(* Logix 5000 project; controller FRCFMS vendor 1 type 14 code 150 rev 33.11; software revision 33.00; part 3 of 3 *)
(* tags used below, declared in another part *)
   CMD_END : DINT;
   CMD_IN : DINT;
   CMD_LEN : DINT;
   CMD_LEN1 : INT;
   CMD_LEN2 : INT;
   CMD_START : DINT;
   Conn_Open : BOOL[32];
   EX_CMD : INT;
   EX_CODE : INT;
   MB_Resp_Data : STR_462;
   Modbus_Byte_cnt : INT;
   Modbus_Cmd_String : STR_462;
   Modbus_Ret_CMD : STRING;
   Modbus_Ret_len : STRING;
   Next_Write : BOOL[32];
   ONS : BOOL[64];
   ONS_B : BOOL[32];
   ONS_ERR : BOOL[32];
   RG_4x_Pos : DINT;
   RW_Instance : INT[20];
   RW_Select : DINT;
   String_Pos : INT;
   Valid : BOOL[32];
   Valid_CMD : BOOL[32];
   Valid_End : BOOL;
   Valid_Len : BOOL;
   Valid_Len_16 : BOOL;
   Valid_Start_Addr : BOOL;
   MBTI_Read_Data_MSG_00 : MESSAGE;
   MBTI_Read_Data_MSG_01 : MESSAGE;
   MBTI_Read_Data_MSG_02 : MESSAGE;
   MBTI_Read_Data_MSG_03 : MESSAGE;
   MBTI_Read_Data_MSG_04 : MESSAGE;
   MBTI_Read_Data_MSG_05 : MESSAGE;
   MBTI_Read_Data_MSG_06 : MESSAGE;
   MBTI_Read_Data_MSG_07 : MESSAGE;
   MBTI_Read_Data_MSG_08 : MESSAGE;
   MBTI_Read_Data_MSG_09 : MESSAGE;
   MBTI_Read_Done : BOOL[32];
   MBTI_Read_Resp : READ_RESP_STR[10];
   MBTI_Write_Data_MSG_00 : MESSAGE;
   MBTI_Write_Data_MSG_01 : MESSAGE;
   MBTI_Write_Data_MSG_02 : MESSAGE;
   MBTI_Write_Data_MSG_03 : MESSAGE;
   MBTI_Write_Data_MSG_04 : MESSAGE;
   MBTI_Write_Data_MSG_05 : MESSAGE;
   MBTI_Write_Data_MSG_06 : MESSAGE;
   MBTI_Write_Data_MSG_07 : MESSAGE;
   MBTI_Write_Data_MSG_08 : MESSAGE;
   MBTI_Write_Data_MSG_09 : MESSAGE;
   MBTI_Write_Data_Out : WRT_DATA[10];
   MBTU_MB_4xx : INT[100];
(* ModbusSlaveTCP, continued *)

ROUTINE SUB_Resp_Str_WORD   (* ladder *)
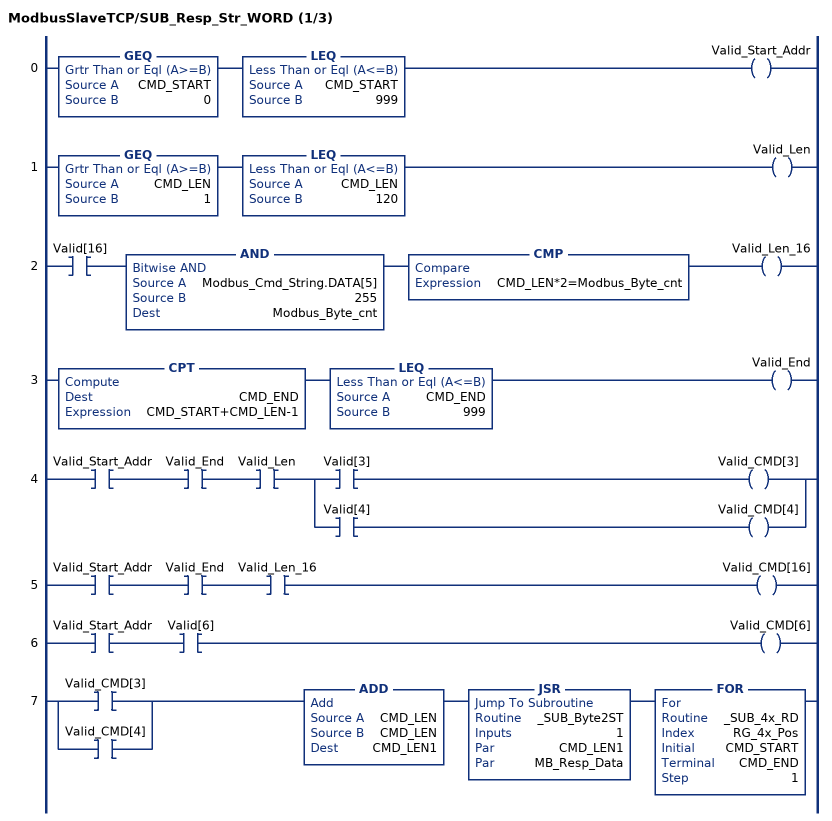
   0: GEQ(CMD_START,0)LEQ(CMD_START,999)OTE(Valid_Start_Addr);
   1: GEQ(CMD_LEN,1)LEQ(CMD_LEN,120)OTE(Valid_Len);
   2: XIC(Valid[16])AND(Modbus_Cmd_String.DATA[5],255,Modbus_Byte_cnt)CMP(CMD_LEN*2=Modbus_Byte_cnt)OTE(Valid_Len_16);
   3: CPT(CMD_END,CMD_START+CMD_LEN-1)LEQ(CMD_END,999)OTE(Valid_End);
   4: XIC(Valid_Start_Addr)XIC(Valid_End)XIC(Valid_Len)[XIC(Valid[3]) OTE(Valid_CMD[3]) ,XIC(Valid[4]) OTE(Valid_CMD[4]) ];
   5: XIC(Valid_Start_Addr)XIC(Valid_End)XIC(Valid_Len_16)OTE(Valid_CMD[16]);
   6: XIC(Valid_Start_Addr)XIC(Valid[6])OTE(Valid_CMD[6]);
   7: [XIC(Valid_CMD[3]) ,XIC(Valid_CMD[4]) ]ADD(CMD_LEN,CMD_LEN,CMD_LEN1)JSR(_SUB_Byte2ST,1,CMD_LEN1,MB_Resp_Data)FOR(_SUB_4x_RD,RG_4x_Pos,CMD_START,CMD_END,1);
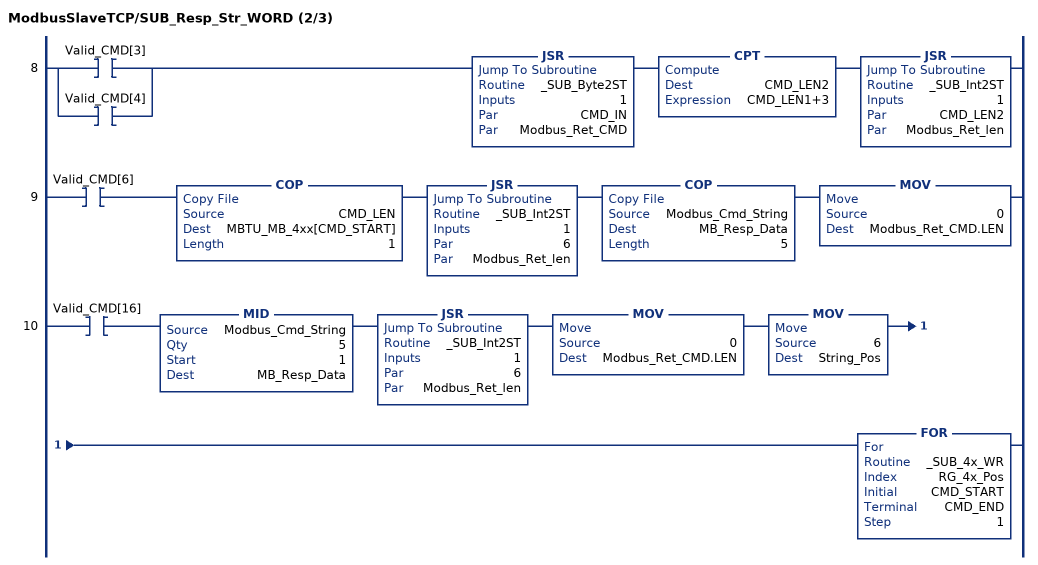
   8: [XIC(Valid_CMD[3]) ,XIC(Valid_CMD[4]) ]JSR(_SUB_Byte2ST,1,CMD_IN,Modbus_Ret_CMD)CPT(CMD_LEN2,CMD_LEN1+3)JSR(_SUB_Int2ST,1,CMD_LEN2,Modbus_Ret_len);
   9: XIC(Valid_CMD[6])COP(CMD_LEN,MBTU_MB_4xx[CMD_START],1)JSR(_SUB_Int2ST,1,6,Modbus_Ret_len)COP(Modbus_Cmd_String,MB_Resp_Data,5)MOV(0,Modbus_Ret_CMD.LEN);
   10: XIC(Valid_CMD[16])MID(Modbus_Cmd_String,5,1,MB_Resp_Data)JSR(_SUB_Int2ST,1,6,Modbus_Ret_len)MOV(0,Modbus_Ret_CMD.LEN)MOV(6,String_Pos)FOR(_SUB_4x_WR,RG_4x_Pos,CMD_START,CMD_END,1);
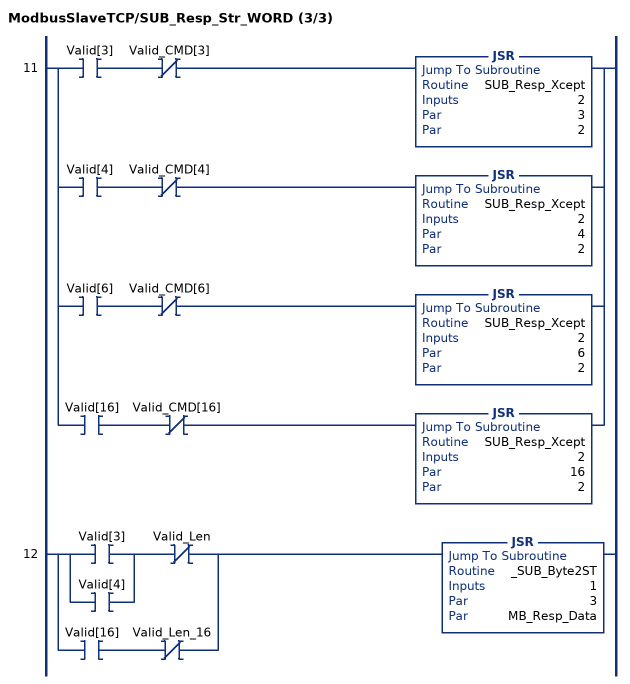
   11: [XIC(Valid[3]) XIO(Valid_CMD[3]) JSR(SUB_Resp_Xcept,2,3,2) ,XIC(Valid[4]) XIO(Valid_CMD[4]) JSR(SUB_Resp_Xcept,2,4,2) ,XIC(Valid[6]) XIO(Valid_CMD[6]) JSR(SUB_Resp_Xcept,2,6,2) ,XIC(Valid[16]) XIO(Valid_CMD[16]) JSR(SUB_Resp_Xcept,2,16,2) ];
   12: [[XIC(Valid[3]) ,XIC(Valid[4]) ] XIO(Valid_Len) ,XIC(Valid[16]) XIO(Valid_Len_16) ]JSR(_SUB_Byte2ST,1,3,MB_Resp_Data);
END_ROUTINE

ROUTINE SUB_Resp_Xcept   (* ladder *)
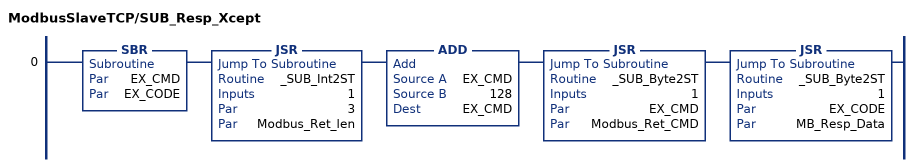
   0: SBR(EX_CMD,EX_CODE)JSR(_SUB_Int2ST,1,3,Modbus_Ret_len)ADD(EX_CMD,128,EX_CMD)JSR(_SUB_Byte2ST,1,EX_CMD,Modbus_Ret_CMD)JSR(_SUB_Byte2ST,1,EX_CODE,MB_Resp_Data);
END_ROUTINE

ROUTINE SUB_RW_Messages   (* ladder *)
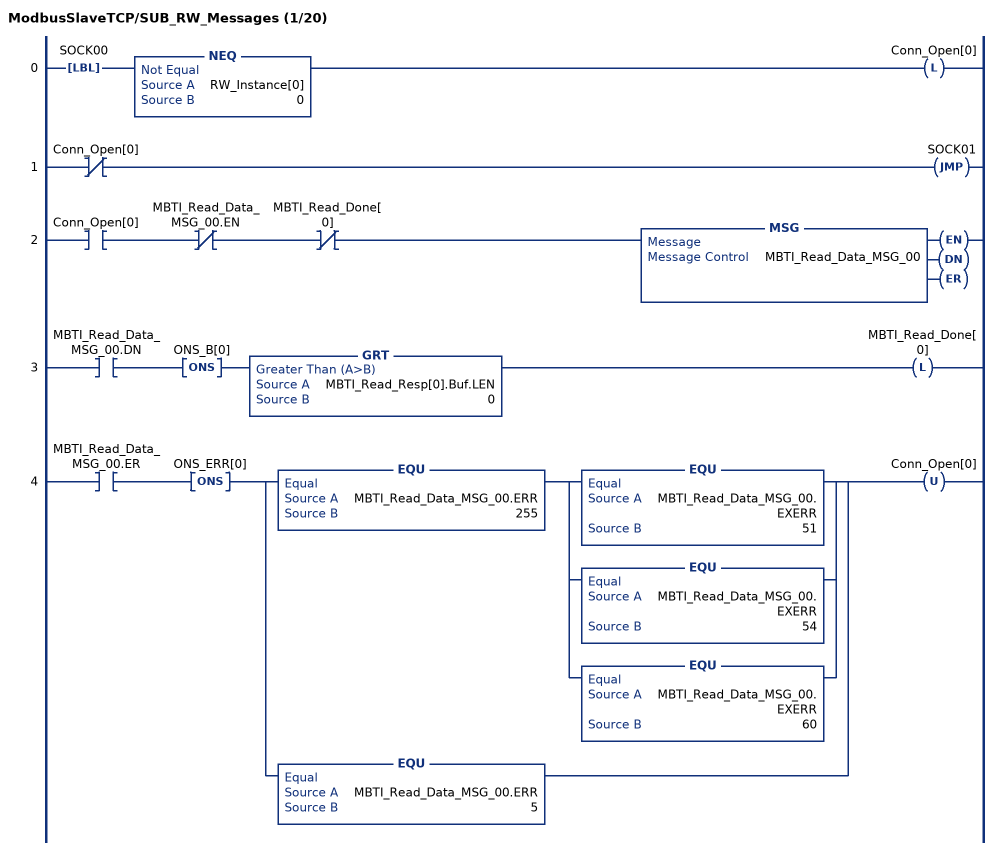
   0: LBL(SOCK00)NEQ(RW_Instance[0],0)OTL(Conn_Open[0]);
   1: XIO(Conn_Open[0])JMP(SOCK01);
   2: XIC(Conn_Open[0])XIO(MBTI_Read_Data_MSG_00.EN)XIO(MBTI_Read_Done[0])MSG(MBTI_Read_Data_MSG_00);
   3: XIC(MBTI_Read_Data_MSG_00.DN)ONS(ONS_B[0])GRT(MBTI_Read_Resp[0].Buf.LEN,0)OTL(MBTI_Read_Done[0]);
   4: XIC(MBTI_Read_Data_MSG_00.ER)ONS(ONS_ERR[0])[EQU(MBTI_Read_Data_MSG_00.ERR,255) [EQU(MBTI_Read_Data_MSG_00.EXERR,51) ,EQU(MBTI_Read_Data_MSG_00.EXERR,54) ,EQU(MBTI_Read_Data_MSG_00.EXERR,60) ] ,EQU(MBTI_Read_Data_MSG_00.ERR,5) ]OTU(Conn_Open[0]);
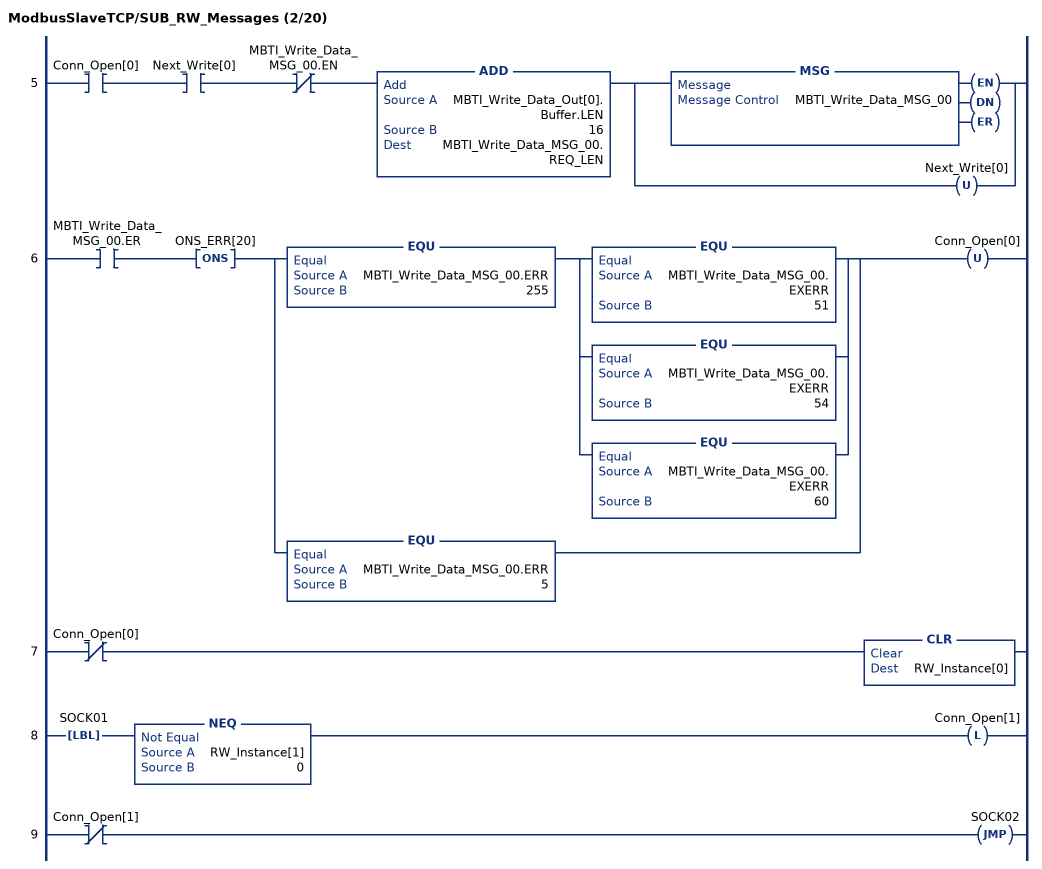
   5: XIC(Conn_Open[0])XIC(Next_Write[0])XIO(MBTI_Write_Data_MSG_00.EN)ADD(MBTI_Write_Data_Out[0].Buffer.LEN,16,MBTI_Write_Data_MSG_00.REQ_LEN)[MSG(MBTI_Write_Data_MSG_00) ,OTU(Next_Write[0]) ];
   6: XIC(MBTI_Write_Data_MSG_00.ER)ONS(ONS_ERR[20])[EQU(MBTI_Write_Data_MSG_00.ERR,255) [EQU(MBTI_Write_Data_MSG_00.EXERR,51) ,EQU(MBTI_Write_Data_MSG_00.EXERR,54) ,EQU(MBTI_Write_Data_MSG_00.EXERR,60) ] ,EQU(MBTI_Write_Data_MSG_00.ERR,5) ]OTU(Conn_Open[0]);
   7: XIO(Conn_Open[0])CLR(RW_Instance[0]);
   8: LBL(SOCK01)NEQ(RW_Instance[1],0)OTL(Conn_Open[1]);
   9: XIO(Conn_Open[1])JMP(SOCK02);
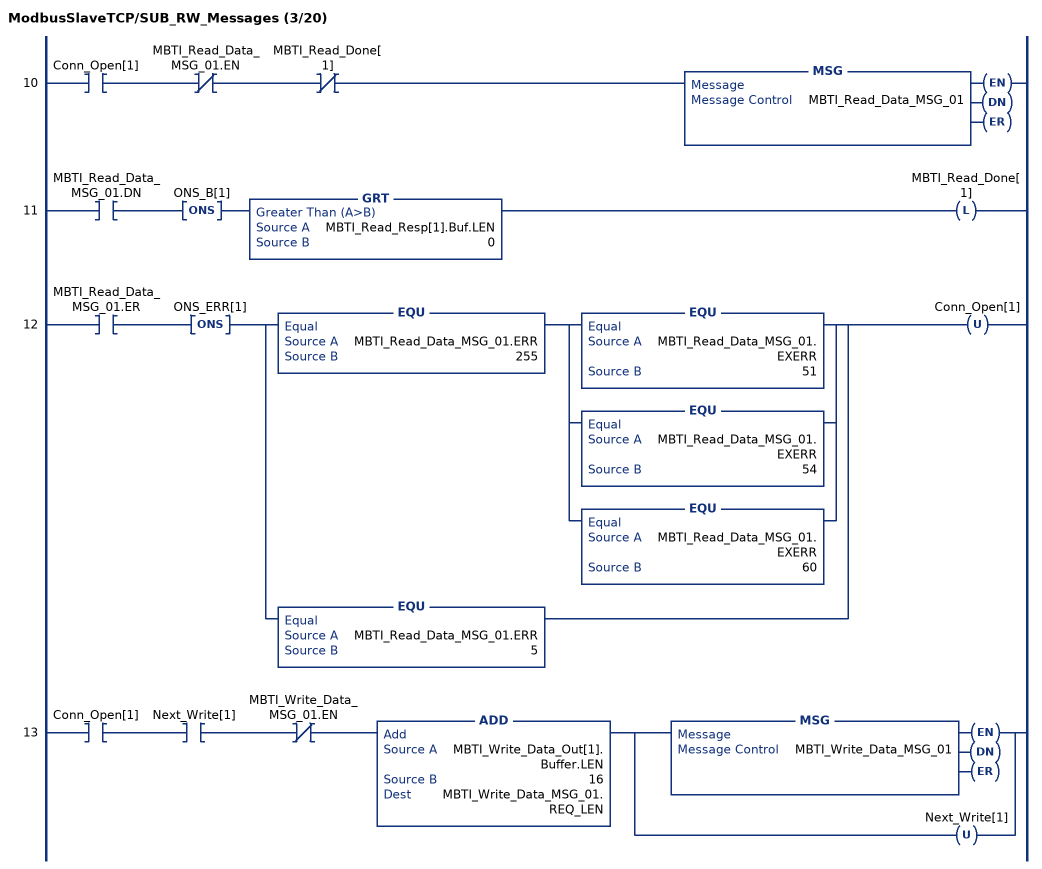
   10: XIC(Conn_Open[1])XIO(MBTI_Read_Data_MSG_01.EN)XIO(MBTI_Read_Done[1])MSG(MBTI_Read_Data_MSG_01);
   11: XIC(MBTI_Read_Data_MSG_01.DN)ONS(ONS_B[1])GRT(MBTI_Read_Resp[1].Buf.LEN,0)OTL(MBTI_Read_Done[1]);
   12: XIC(MBTI_Read_Data_MSG_01.ER)ONS(ONS_ERR[1])[EQU(MBTI_Read_Data_MSG_01.ERR,255) [EQU(MBTI_Read_Data_MSG_01.EXERR,51) ,EQU(MBTI_Read_Data_MSG_01.EXERR,54) ,EQU(MBTI_Read_Data_MSG_01.EXERR,60) ] ,EQU(MBTI_Read_Data_MSG_01.ERR,5) ]OTU(Conn_Open[1]);
   13: XIC(Conn_Open[1])XIC(Next_Write[1])XIO(MBTI_Write_Data_MSG_01.EN)ADD(MBTI_Write_Data_Out[1].Buffer.LEN,16,MBTI_Write_Data_MSG_01.REQ_LEN)[MSG(MBTI_Write_Data_MSG_01) ,OTU(Next_Write[1]) ];
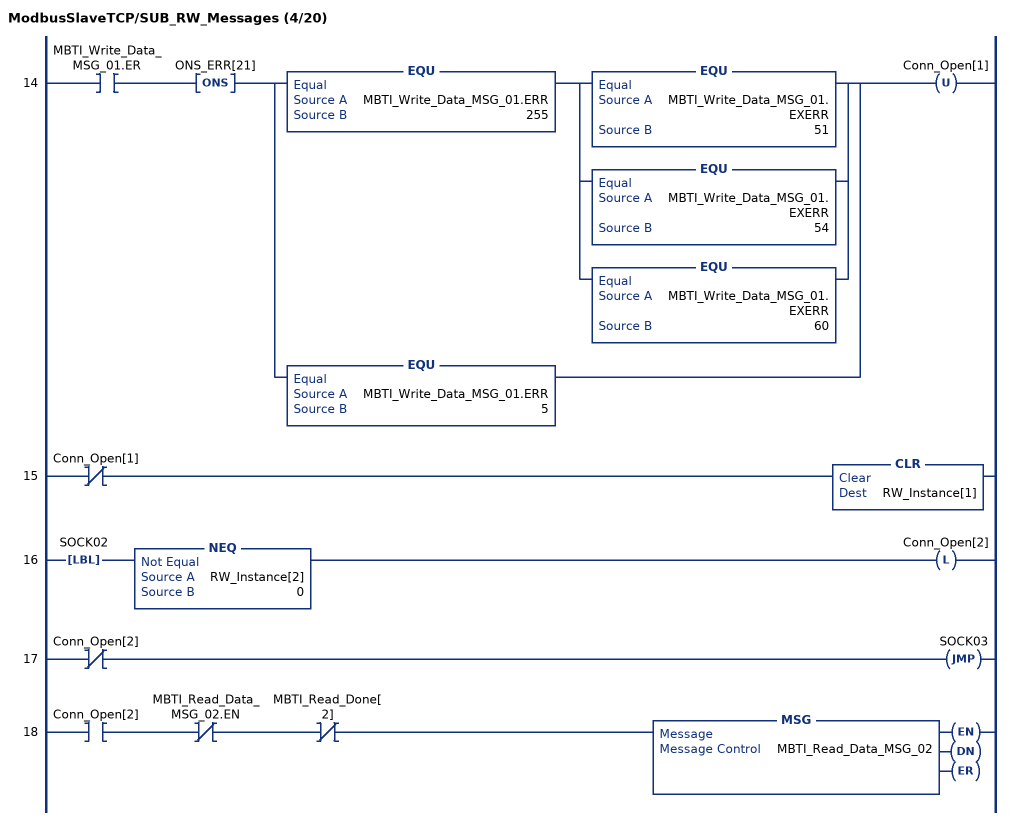
   14: XIC(MBTI_Write_Data_MSG_01.ER)ONS(ONS_ERR[21])[EQU(MBTI_Write_Data_MSG_01.ERR,255) [EQU(MBTI_Write_Data_MSG_01.EXERR,51) ,EQU(MBTI_Write_Data_MSG_01.EXERR,54) ,EQU(MBTI_Write_Data_MSG_01.EXERR,60) ] ,EQU(MBTI_Write_Data_MSG_01.ERR,5) ]OTU(Conn_Open[1]);
   15: XIO(Conn_Open[1])CLR(RW_Instance[1]);
   16: LBL(SOCK02)NEQ(RW_Instance[2],0)OTL(Conn_Open[2]);
   17: XIO(Conn_Open[2])JMP(SOCK03);
   18: XIC(Conn_Open[2])XIO(MBTI_Read_Data_MSG_02.EN)XIO(MBTI_Read_Done[2])MSG(MBTI_Read_Data_MSG_02);
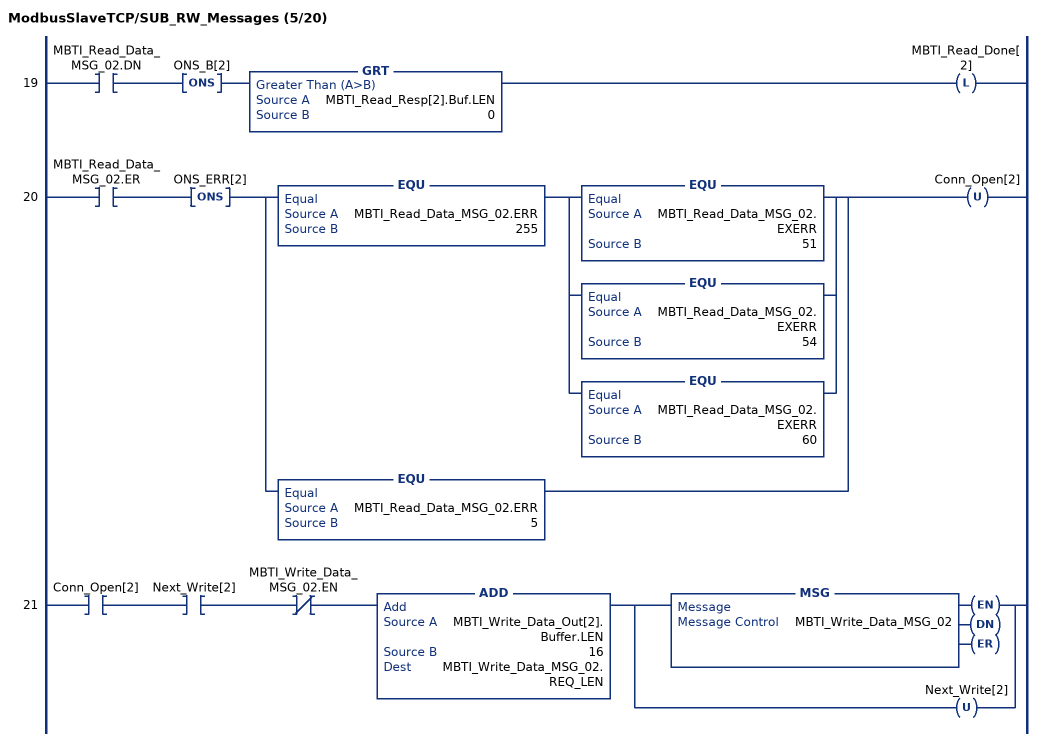
   19: XIC(MBTI_Read_Data_MSG_02.DN)ONS(ONS_B[2])GRT(MBTI_Read_Resp[2].Buf.LEN,0)OTL(MBTI_Read_Done[2]);
   20: XIC(MBTI_Read_Data_MSG_02.ER)ONS(ONS_ERR[2])[EQU(MBTI_Read_Data_MSG_02.ERR,255) [EQU(MBTI_Read_Data_MSG_02.EXERR,51) ,EQU(MBTI_Read_Data_MSG_02.EXERR,54) ,EQU(MBTI_Read_Data_MSG_02.EXERR,60) ] ,EQU(MBTI_Read_Data_MSG_02.ERR,5) ]OTU(Conn_Open[2]);
   21: XIC(Conn_Open[2])XIC(Next_Write[2])XIO(MBTI_Write_Data_MSG_02.EN)ADD(MBTI_Write_Data_Out[2].Buffer.LEN,16,MBTI_Write_Data_MSG_02.REQ_LEN)[MSG(MBTI_Write_Data_MSG_02) ,OTU(Next_Write[2]) ];
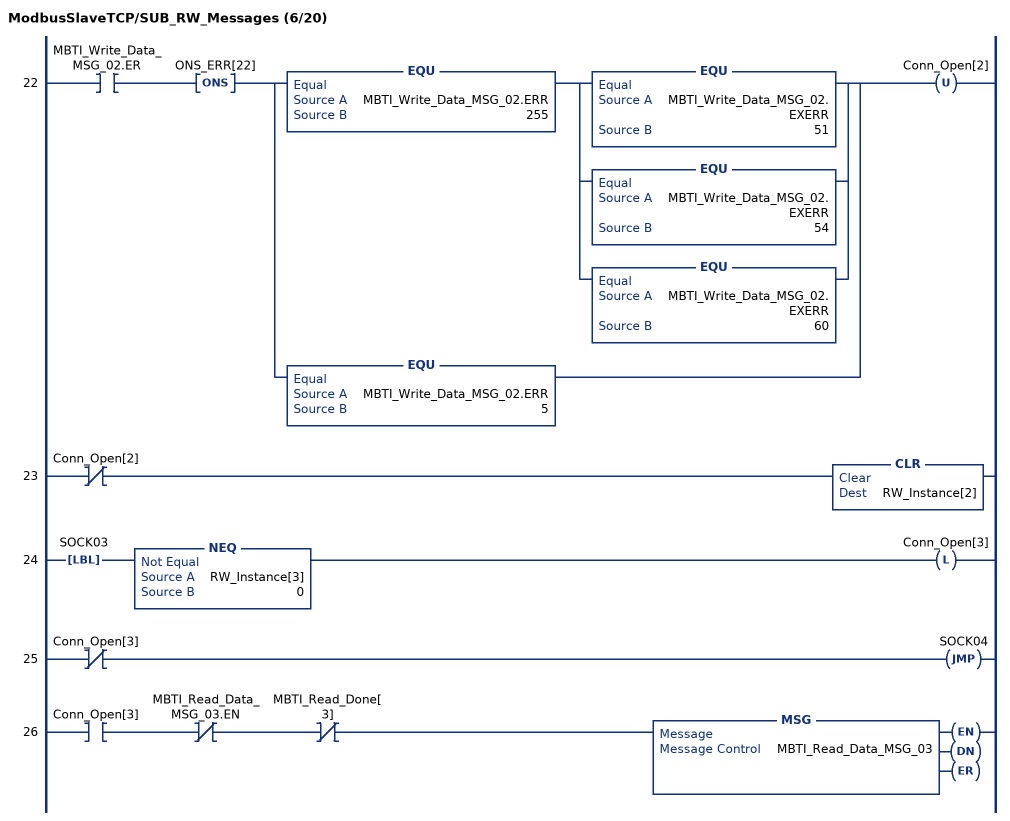
   22: XIC(MBTI_Write_Data_MSG_02.ER)ONS(ONS_ERR[22])[EQU(MBTI_Write_Data_MSG_02.ERR,255) [EQU(MBTI_Write_Data_MSG_02.EXERR,51) ,EQU(MBTI_Write_Data_MSG_02.EXERR,54) ,EQU(MBTI_Write_Data_MSG_02.EXERR,60) ] ,EQU(MBTI_Write_Data_MSG_02.ERR,5) ]OTU(Conn_Open[2]);
   23: XIO(Conn_Open[2])CLR(RW_Instance[2]);
   24: LBL(SOCK03)NEQ(RW_Instance[3],0)OTL(Conn_Open[3]);
   25: XIO(Conn_Open[3])JMP(SOCK04);
   26: XIC(Conn_Open[3])XIO(MBTI_Read_Data_MSG_03.EN)XIO(MBTI_Read_Done[3])MSG(MBTI_Read_Data_MSG_03);
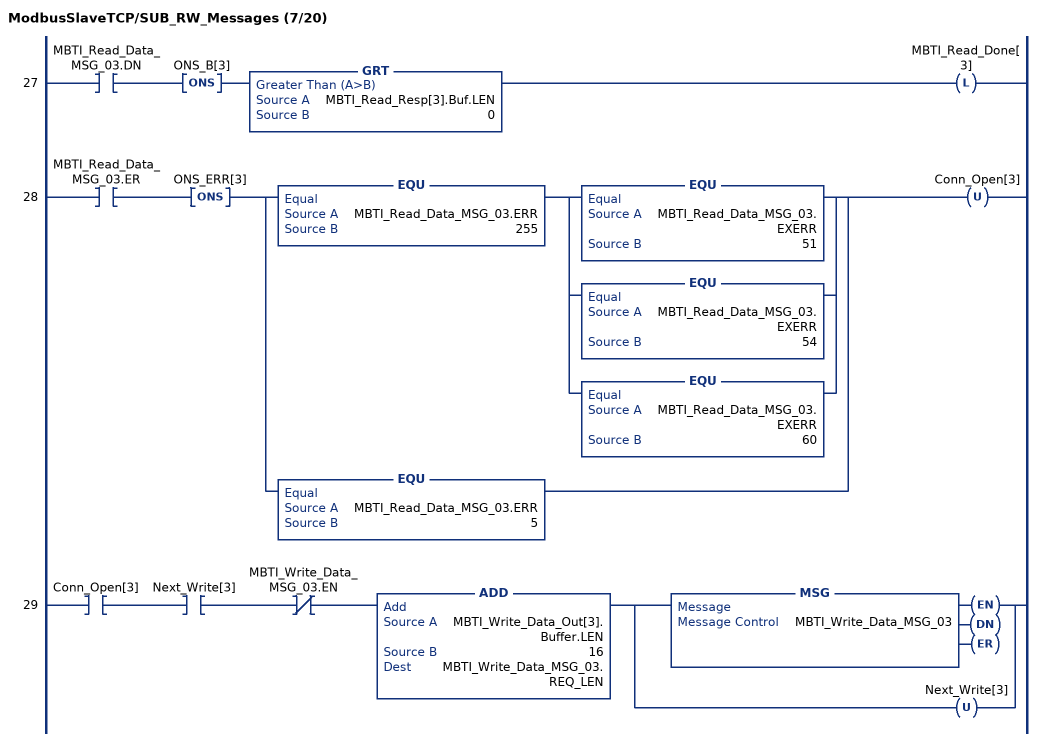
   27: XIC(MBTI_Read_Data_MSG_03.DN)ONS(ONS_B[3])GRT(MBTI_Read_Resp[3].Buf.LEN,0)OTL(MBTI_Read_Done[3]);
   28: XIC(MBTI_Read_Data_MSG_03.ER)ONS(ONS_ERR[3])[EQU(MBTI_Read_Data_MSG_03.ERR,255) [EQU(MBTI_Read_Data_MSG_03.EXERR,51) ,EQU(MBTI_Read_Data_MSG_03.EXERR,54) ,EQU(MBTI_Read_Data_MSG_03.EXERR,60) ] ,EQU(MBTI_Read_Data_MSG_03.ERR,5) ]OTU(Conn_Open[3]);
   29: XIC(Conn_Open[3])XIC(Next_Write[3])XIO(MBTI_Write_Data_MSG_03.EN)ADD(MBTI_Write_Data_Out[3].Buffer.LEN,16,MBTI_Write_Data_MSG_03.REQ_LEN)[MSG(MBTI_Write_Data_MSG_03) ,OTU(Next_Write[3]) ];
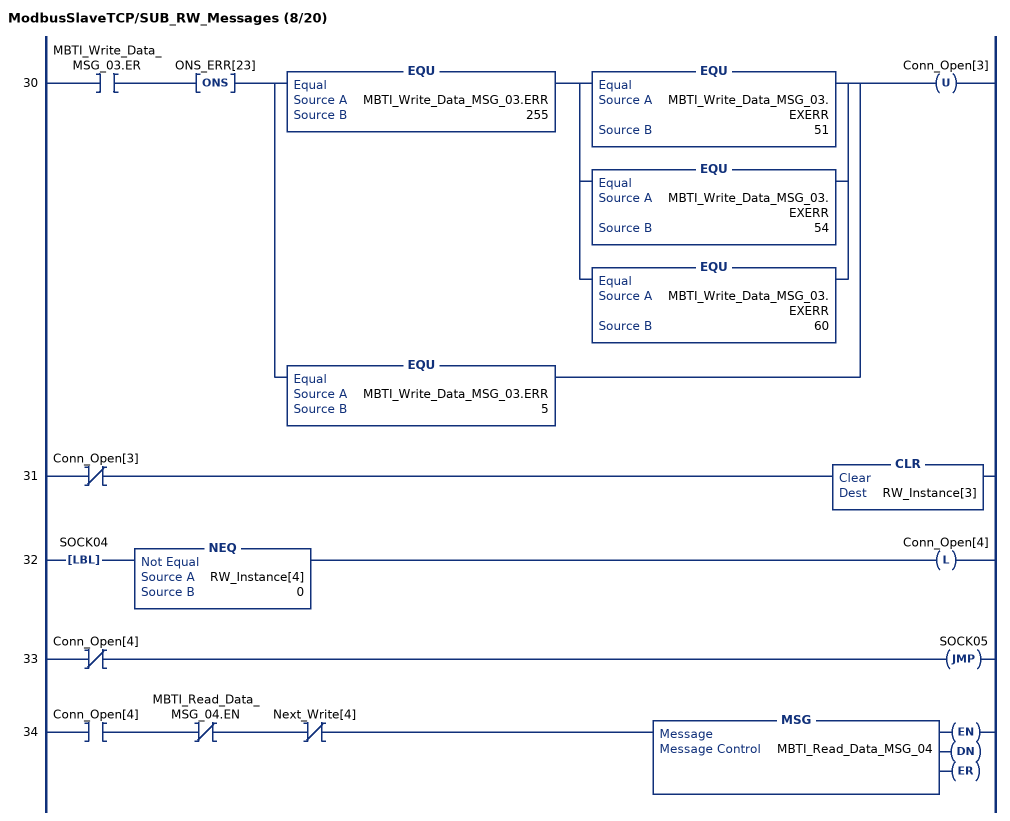
   30: XIC(MBTI_Write_Data_MSG_03.ER)ONS(ONS_ERR[23])[EQU(MBTI_Write_Data_MSG_03.ERR,255) [EQU(MBTI_Write_Data_MSG_03.EXERR,51) ,EQU(MBTI_Write_Data_MSG_03.EXERR,54) ,EQU(MBTI_Write_Data_MSG_03.EXERR,60) ] ,EQU(MBTI_Write_Data_MSG_03.ERR,5) ]OTU(Conn_Open[3]);
   31: XIO(Conn_Open[3])CLR(RW_Instance[3]);
   32: LBL(SOCK04)NEQ(RW_Instance[4],0)OTL(Conn_Open[4]);
   33: XIO(Conn_Open[4])JMP(SOCK05);
   34: XIC(Conn_Open[4])XIO(MBTI_Read_Data_MSG_04.EN)XIO(Next_Write[4])MSG(MBTI_Read_Data_MSG_04);
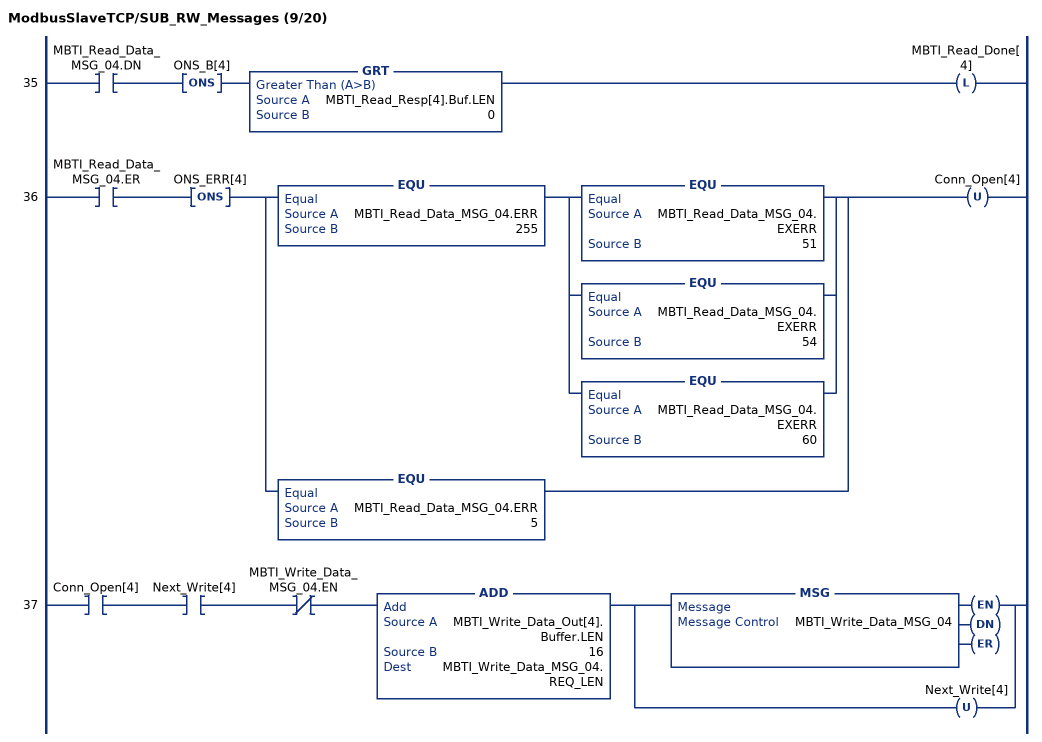
   35: XIC(MBTI_Read_Data_MSG_04.DN)ONS(ONS_B[4])GRT(MBTI_Read_Resp[4].Buf.LEN,0)OTL(MBTI_Read_Done[4]);
   36: XIC(MBTI_Read_Data_MSG_04.ER)ONS(ONS_ERR[4])[EQU(MBTI_Read_Data_MSG_04.ERR,255) [EQU(MBTI_Read_Data_MSG_04.EXERR,51) ,EQU(MBTI_Read_Data_MSG_04.EXERR,54) ,EQU(MBTI_Read_Data_MSG_04.EXERR,60) ] ,EQU(MBTI_Read_Data_MSG_04.ERR,5) ]OTU(Conn_Open[4]);
   37: XIC(Conn_Open[4])XIC(Next_Write[4])XIO(MBTI_Write_Data_MSG_04.EN)ADD(MBTI_Write_Data_Out[4].Buffer.LEN,16,MBTI_Write_Data_MSG_04.REQ_LEN)[MSG(MBTI_Write_Data_MSG_04) ,OTU(Next_Write[4]) ];
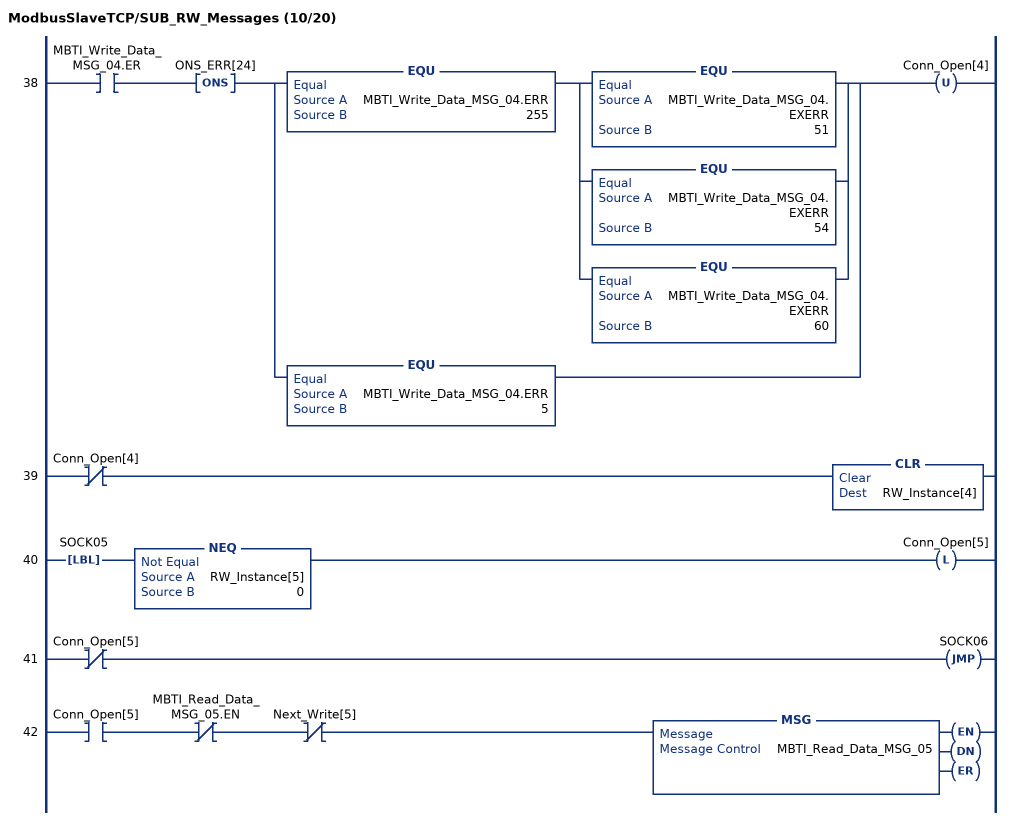
   38: XIC(MBTI_Write_Data_MSG_04.ER)ONS(ONS_ERR[24])[EQU(MBTI_Write_Data_MSG_04.ERR,255) [EQU(MBTI_Write_Data_MSG_04.EXERR,51) ,EQU(MBTI_Write_Data_MSG_04.EXERR,54) ,EQU(MBTI_Write_Data_MSG_04.EXERR,60) ] ,EQU(MBTI_Write_Data_MSG_04.ERR,5) ]OTU(Conn_Open[4]);
   39: XIO(Conn_Open[4])CLR(RW_Instance[4]);
   40: LBL(SOCK05)NEQ(RW_Instance[5],0)OTL(Conn_Open[5]);
   41: XIO(Conn_Open[5])JMP(SOCK06);
   42: XIC(Conn_Open[5])XIO(MBTI_Read_Data_MSG_05.EN)XIO(Next_Write[5])MSG(MBTI_Read_Data_MSG_05);
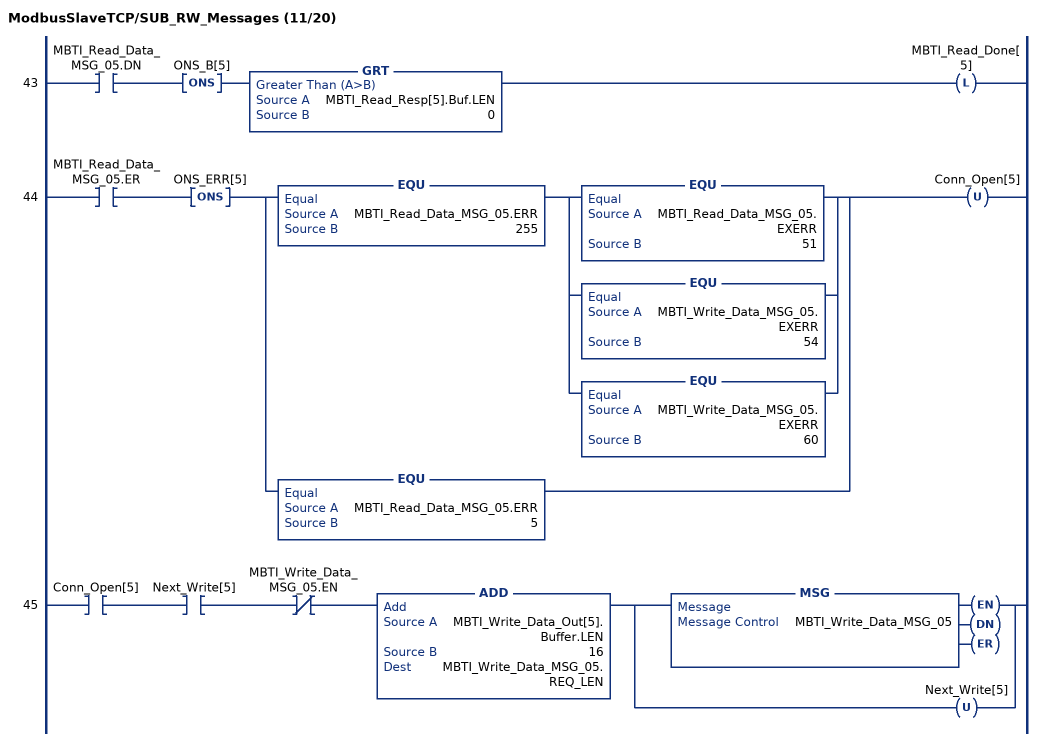
   43: XIC(MBTI_Read_Data_MSG_05.DN)ONS(ONS_B[5])GRT(MBTI_Read_Resp[5].Buf.LEN,0)OTL(MBTI_Read_Done[5]);
   44: XIC(MBTI_Read_Data_MSG_05.ER)ONS(ONS_ERR[5])[EQU(MBTI_Read_Data_MSG_05.ERR,255) [EQU(MBTI_Read_Data_MSG_05.EXERR,51) ,EQU(MBTI_Write_Data_MSG_05.EXERR,54) ,EQU(MBTI_Write_Data_MSG_05.EXERR,60) ] ,EQU(MBTI_Read_Data_MSG_05.ERR,5) ]OTU(Conn_Open[5]);
   45: XIC(Conn_Open[5])XIC(Next_Write[5])XIO(MBTI_Write_Data_MSG_05.EN)ADD(MBTI_Write_Data_Out[5].Buffer.LEN,16,MBTI_Write_Data_MSG_05.REQ_LEN)[MSG(MBTI_Write_Data_MSG_05) ,OTU(Next_Write[5]) ];
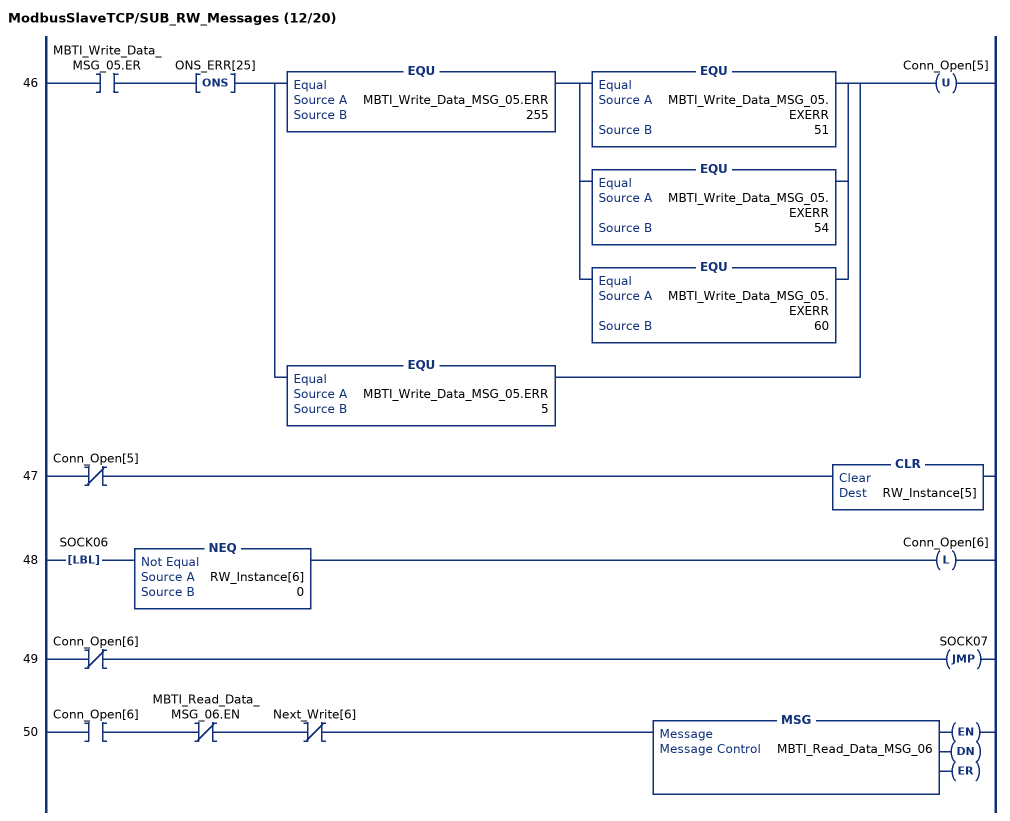
   46: XIC(MBTI_Write_Data_MSG_05.ER)ONS(ONS_ERR[25])[EQU(MBTI_Write_Data_MSG_05.ERR,255) [EQU(MBTI_Write_Data_MSG_05.EXERR,51) ,EQU(MBTI_Write_Data_MSG_05.EXERR,54) ,EQU(MBTI_Write_Data_MSG_05.EXERR,60) ] ,EQU(MBTI_Write_Data_MSG_05.ERR,5) ]OTU(Conn_Open[5]);
   47: XIO(Conn_Open[5])CLR(RW_Instance[5]);
   48: LBL(SOCK06)NEQ(RW_Instance[6],0)OTL(Conn_Open[6]);
   49: XIO(Conn_Open[6])JMP(SOCK07);
   50: XIC(Conn_Open[6])XIO(MBTI_Read_Data_MSG_06.EN)XIO(Next_Write[6])MSG(MBTI_Read_Data_MSG_06);
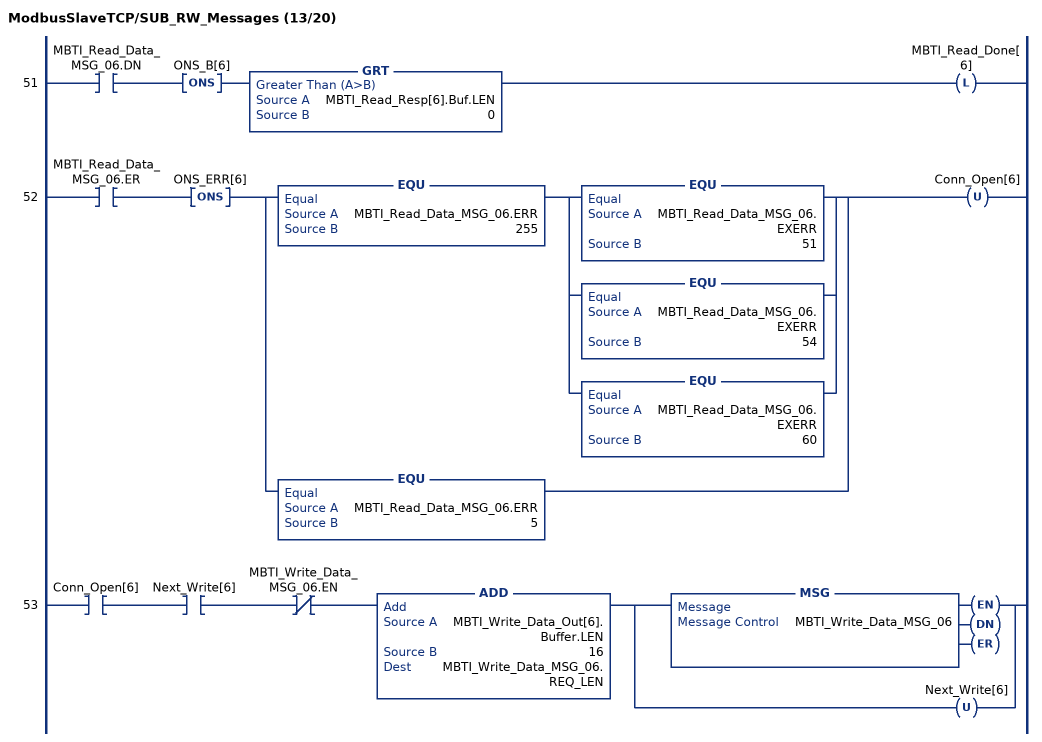
   51: XIC(MBTI_Read_Data_MSG_06.DN)ONS(ONS_B[6])GRT(MBTI_Read_Resp[6].Buf.LEN,0)OTL(MBTI_Read_Done[6]);
   52: XIC(MBTI_Read_Data_MSG_06.ER)ONS(ONS_ERR[6])[EQU(MBTI_Read_Data_MSG_06.ERR,255) [EQU(MBTI_Read_Data_MSG_06.EXERR,51) ,EQU(MBTI_Read_Data_MSG_06.EXERR,54) ,EQU(MBTI_Read_Data_MSG_06.EXERR,60) ] ,EQU(MBTI_Read_Data_MSG_06.ERR,5) ]OTU(Conn_Open[6]);
   53: XIC(Conn_Open[6])XIC(Next_Write[6])XIO(MBTI_Write_Data_MSG_06.EN)ADD(MBTI_Write_Data_Out[6].Buffer.LEN,16,MBTI_Write_Data_MSG_06.REQ_LEN)[MSG(MBTI_Write_Data_MSG_06) ,OTU(Next_Write[6]) ];
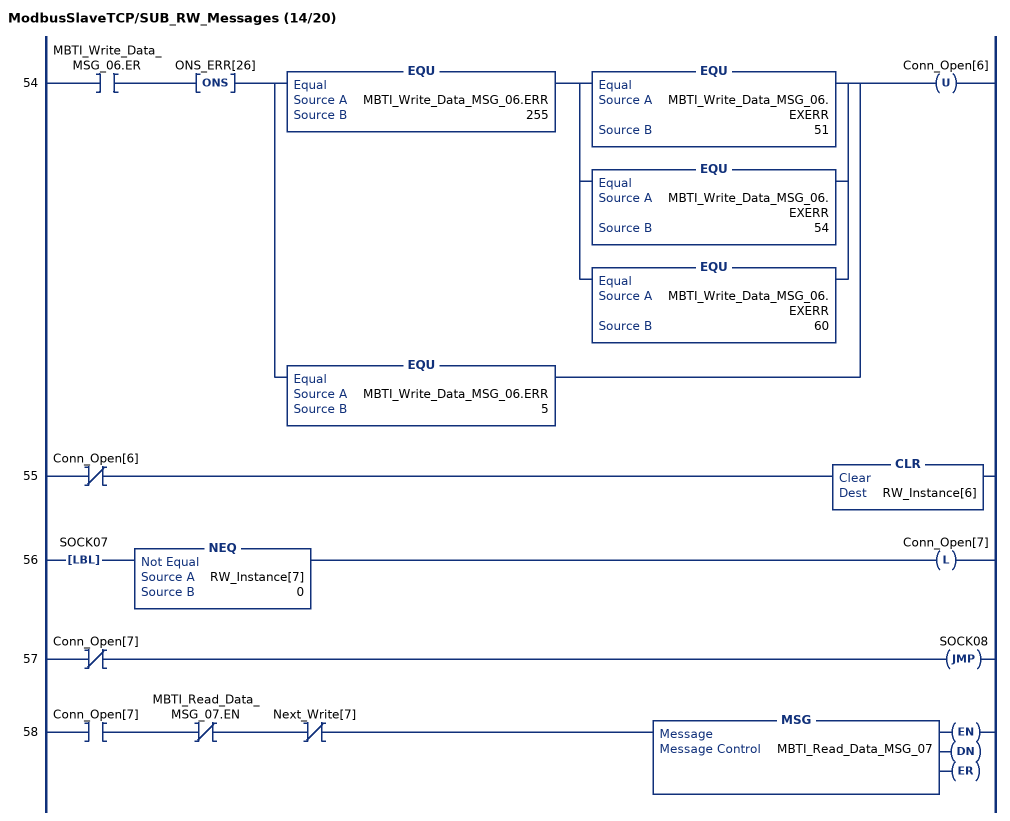
   54: XIC(MBTI_Write_Data_MSG_06.ER)ONS(ONS_ERR[26])[EQU(MBTI_Write_Data_MSG_06.ERR,255) [EQU(MBTI_Write_Data_MSG_06.EXERR,51) ,EQU(MBTI_Write_Data_MSG_06.EXERR,54) ,EQU(MBTI_Write_Data_MSG_06.EXERR,60) ] ,EQU(MBTI_Write_Data_MSG_06.ERR,5) ]OTU(Conn_Open[6]);
   55: XIO(Conn_Open[6])CLR(RW_Instance[6]);
   56: LBL(SOCK07)NEQ(RW_Instance[7],0)OTL(Conn_Open[7]);
   57: XIO(Conn_Open[7])JMP(SOCK08);
   58: XIC(Conn_Open[7])XIO(MBTI_Read_Data_MSG_07.EN)XIO(Next_Write[7])MSG(MBTI_Read_Data_MSG_07);
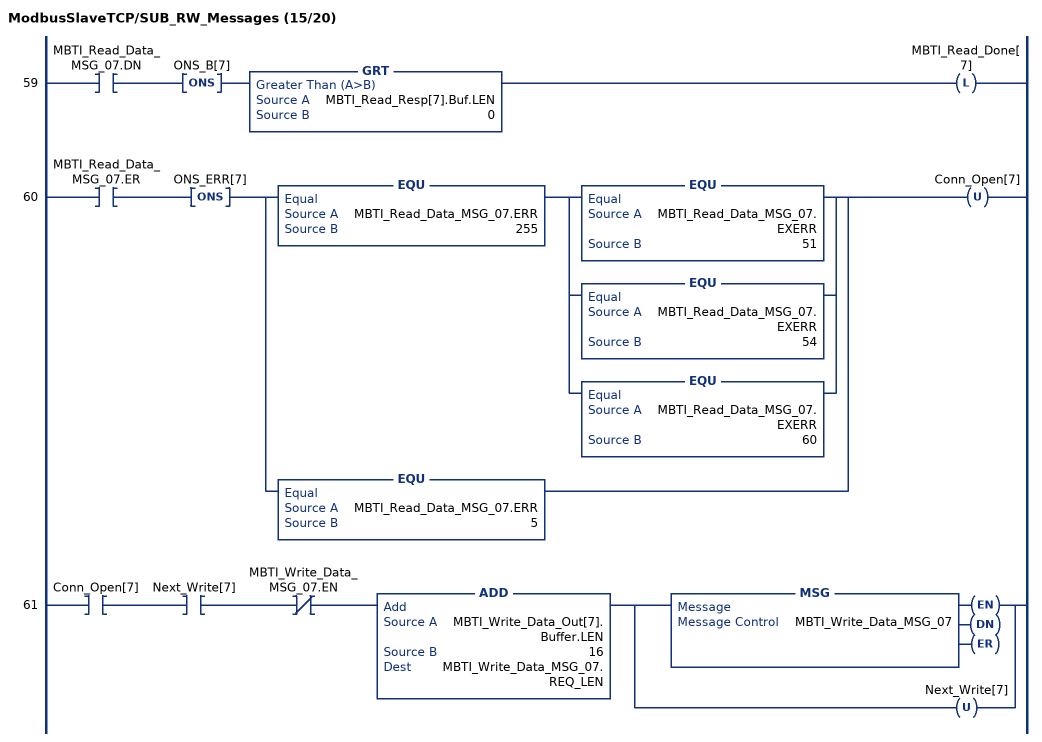
   59: XIC(MBTI_Read_Data_MSG_07.DN)ONS(ONS_B[7])GRT(MBTI_Read_Resp[7].Buf.LEN,0)OTL(MBTI_Read_Done[7]);
   60: XIC(MBTI_Read_Data_MSG_07.ER)ONS(ONS_ERR[7])[EQU(MBTI_Read_Data_MSG_07.ERR,255) [EQU(MBTI_Read_Data_MSG_07.EXERR,51) ,EQU(MBTI_Read_Data_MSG_07.EXERR,54) ,EQU(MBTI_Read_Data_MSG_07.EXERR,60) ] ,EQU(MBTI_Read_Data_MSG_07.ERR,5) ]OTU(Conn_Open[7]);
   61: XIC(Conn_Open[7])XIC(Next_Write[7])XIO(MBTI_Write_Data_MSG_07.EN)ADD(MBTI_Write_Data_Out[7].Buffer.LEN,16,MBTI_Write_Data_MSG_07.REQ_LEN)[MSG(MBTI_Write_Data_MSG_07) ,OTU(Next_Write[7]) ];
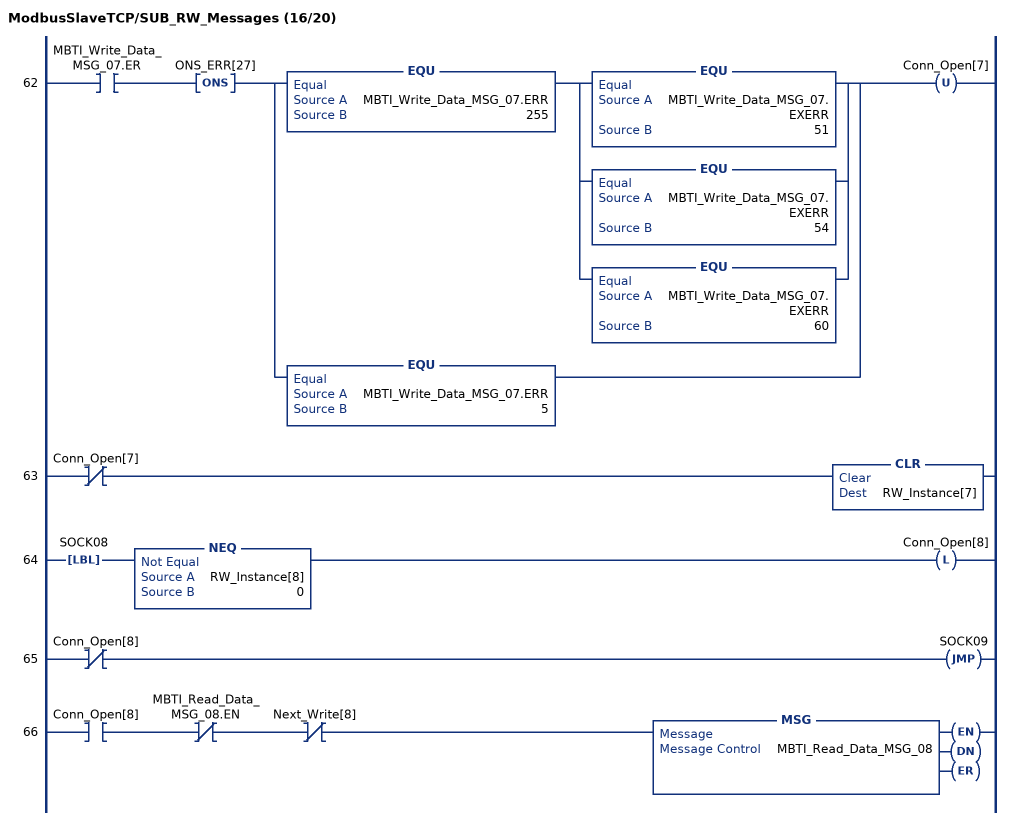
   62: XIC(MBTI_Write_Data_MSG_07.ER)ONS(ONS_ERR[27])[EQU(MBTI_Write_Data_MSG_07.ERR,255) [EQU(MBTI_Write_Data_MSG_07.EXERR,51) ,EQU(MBTI_Write_Data_MSG_07.EXERR,54) ,EQU(MBTI_Write_Data_MSG_07.EXERR,60) ] ,EQU(MBTI_Write_Data_MSG_07.ERR,5) ]OTU(Conn_Open[7]);
   63: XIO(Conn_Open[7])CLR(RW_Instance[7]);
   64: LBL(SOCK08)NEQ(RW_Instance[8],0)OTL(Conn_Open[8]);
   65: XIO(Conn_Open[8])JMP(SOCK09);
   66: XIC(Conn_Open[8])XIO(MBTI_Read_Data_MSG_08.EN)XIO(Next_Write[8])MSG(MBTI_Read_Data_MSG_08);
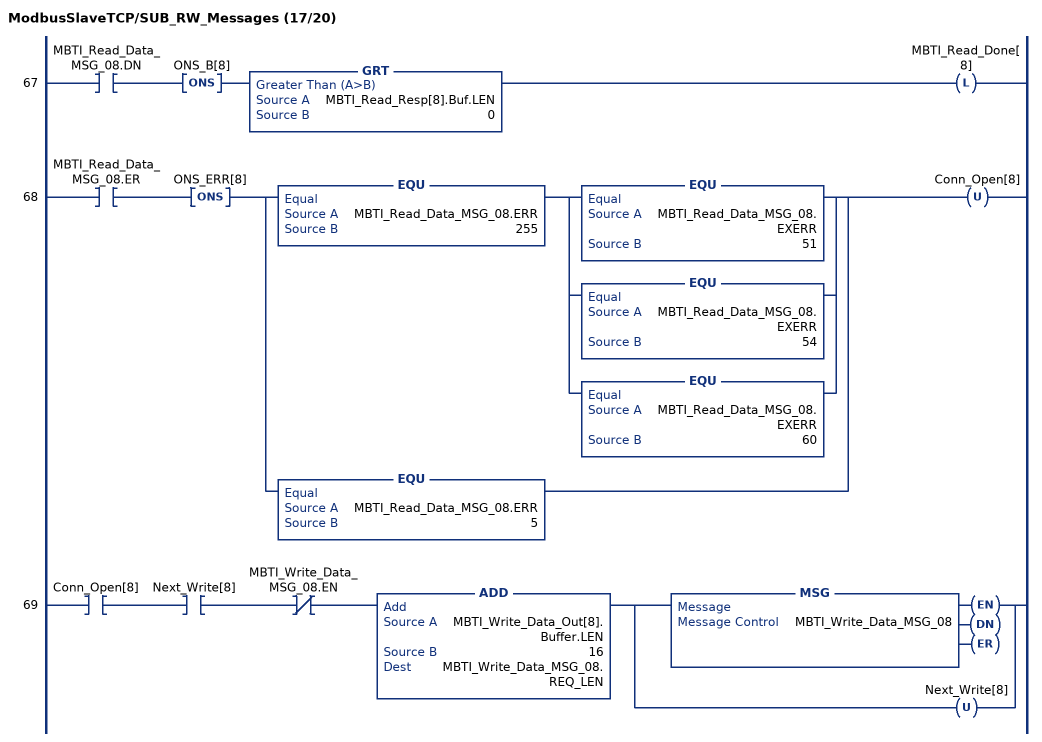
   67: XIC(MBTI_Read_Data_MSG_08.DN)ONS(ONS_B[8])GRT(MBTI_Read_Resp[8].Buf.LEN,0)OTL(MBTI_Read_Done[8]);
   68: XIC(MBTI_Read_Data_MSG_08.ER)ONS(ONS_ERR[8])[EQU(MBTI_Read_Data_MSG_08.ERR,255) [EQU(MBTI_Read_Data_MSG_08.EXERR,51) ,EQU(MBTI_Read_Data_MSG_08.EXERR,54) ,EQU(MBTI_Read_Data_MSG_08.EXERR,60) ] ,EQU(MBTI_Read_Data_MSG_08.ERR,5) ]OTU(Conn_Open[8]);
   69: XIC(Conn_Open[8])XIC(Next_Write[8])XIO(MBTI_Write_Data_MSG_08.EN)ADD(MBTI_Write_Data_Out[8].Buffer.LEN,16,MBTI_Write_Data_MSG_08.REQ_LEN)[MSG(MBTI_Write_Data_MSG_08) ,OTU(Next_Write[8]) ];
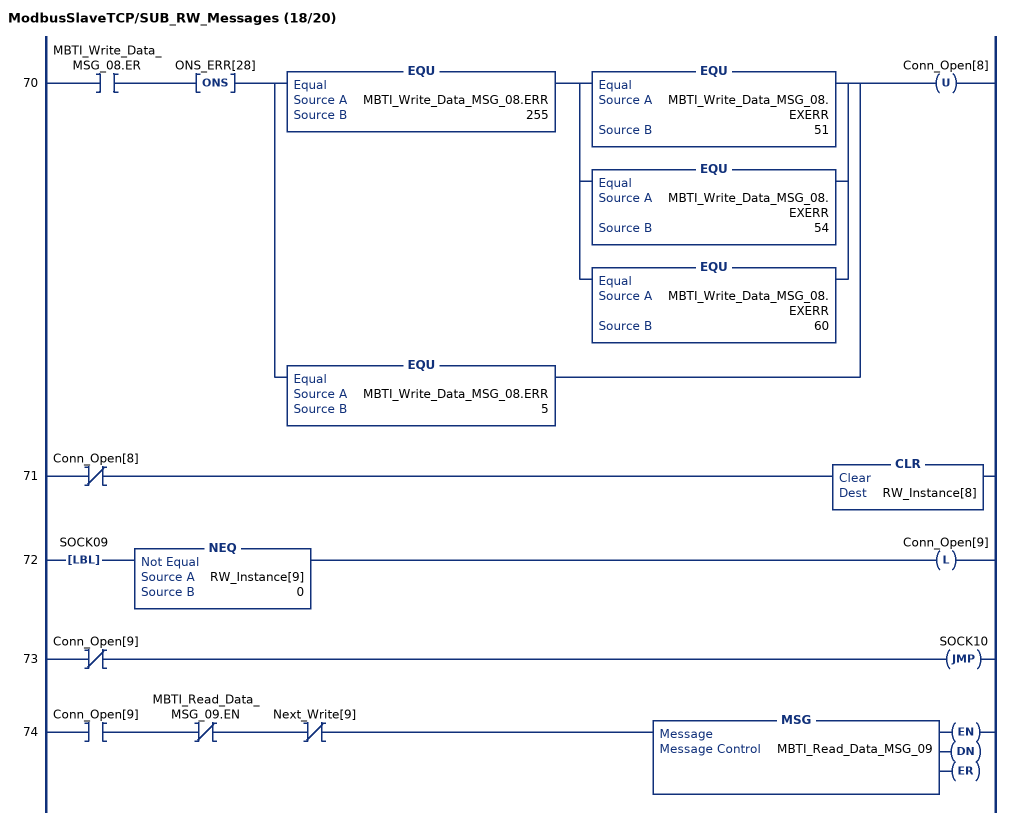
   70: XIC(MBTI_Write_Data_MSG_08.ER)ONS(ONS_ERR[28])[EQU(MBTI_Write_Data_MSG_08.ERR,255) [EQU(MBTI_Write_Data_MSG_08.EXERR,51) ,EQU(MBTI_Write_Data_MSG_08.EXERR,54) ,EQU(MBTI_Write_Data_MSG_08.EXERR,60) ] ,EQU(MBTI_Write_Data_MSG_08.ERR,5) ]OTU(Conn_Open[8]);
   71: XIO(Conn_Open[8])CLR(RW_Instance[8]);
   72: LBL(SOCK09)NEQ(RW_Instance[9],0)OTL(Conn_Open[9]);
   73: XIO(Conn_Open[9])JMP(SOCK10);
   74: XIC(Conn_Open[9])XIO(MBTI_Read_Data_MSG_09.EN)XIO(Next_Write[9])MSG(MBTI_Read_Data_MSG_09);
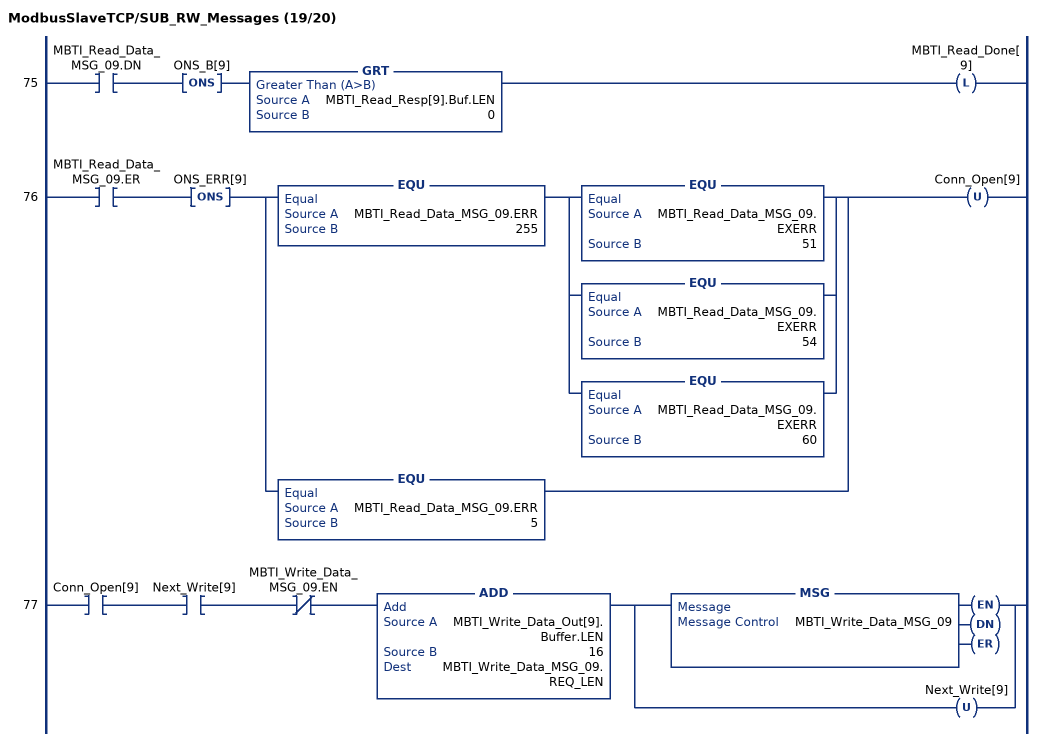
   75: XIC(MBTI_Read_Data_MSG_09.DN)ONS(ONS_B[9])GRT(MBTI_Read_Resp[9].Buf.LEN,0)OTL(MBTI_Read_Done[9]);
   76: XIC(MBTI_Read_Data_MSG_09.ER)ONS(ONS_ERR[9])[EQU(MBTI_Read_Data_MSG_09.ERR,255) [EQU(MBTI_Read_Data_MSG_09.EXERR,51) ,EQU(MBTI_Read_Data_MSG_09.EXERR,54) ,EQU(MBTI_Read_Data_MSG_09.EXERR,60) ] ,EQU(MBTI_Read_Data_MSG_09.ERR,5) ]OTU(Conn_Open[9]);
   77: XIC(Conn_Open[9])XIC(Next_Write[9])XIO(MBTI_Write_Data_MSG_09.EN)ADD(MBTI_Write_Data_Out[9].Buffer.LEN,16,MBTI_Write_Data_MSG_09.REQ_LEN)[MSG(MBTI_Write_Data_MSG_09) ,OTU(Next_Write[9]) ];
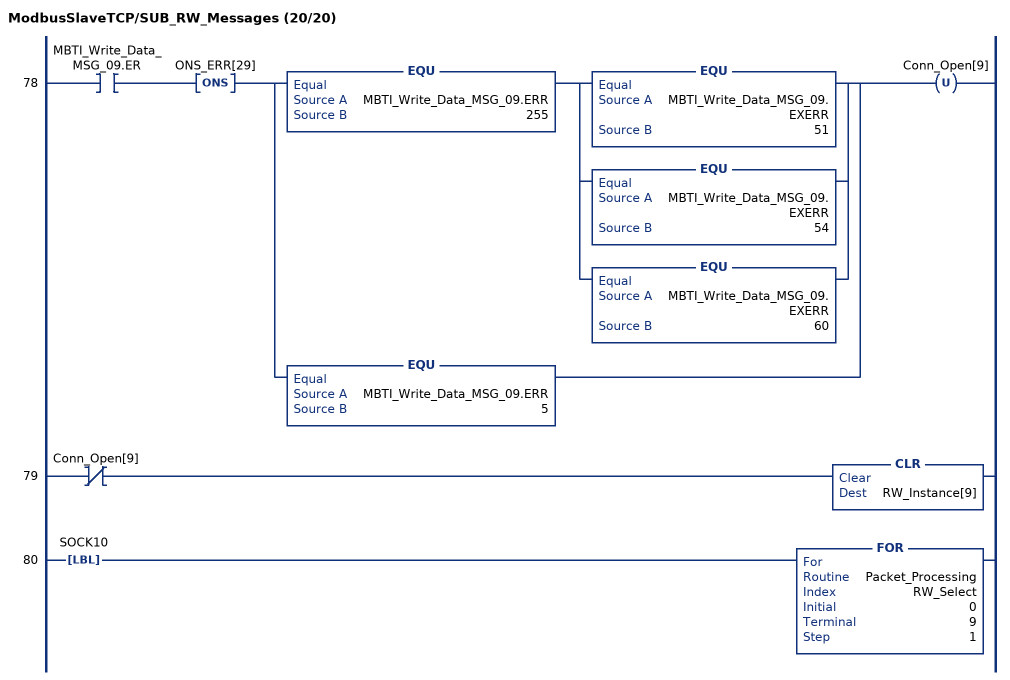
   78: XIC(MBTI_Write_Data_MSG_09.ER)ONS(ONS_ERR[29])[EQU(MBTI_Write_Data_MSG_09.ERR,255) [EQU(MBTI_Write_Data_MSG_09.EXERR,51) ,EQU(MBTI_Write_Data_MSG_09.EXERR,54) ,EQU(MBTI_Write_Data_MSG_09.EXERR,60) ] ,EQU(MBTI_Write_Data_MSG_09.ERR,5) ]OTU(Conn_Open[9]);
   79: XIO(Conn_Open[9])CLR(RW_Instance[9]);
   80: LBL(SOCK10)FOR(Packet_Processing,RW_Select,0,9,1);
END_ROUTINE
END_PROGRAM
